Fanuc KAREL source: CE0115.KL

-- PROVISIONAL review KL for V770-1; original PC SHA256 38c2cadad195cee7491331c5a626b45bc0db98ebdebf5f674fdae5275aeffe66
-- Incomplete behavior may be omitted. Consult companion uncertainty JSON. Do not deploy.
PROGRAM CE0115
%NOLOCKGROUP
-- UNRESOLVED_LOCAL_POOL 6 cells at code offset 94; source declarations unknown
-- DIRECT_LOCAL_WORD_ACCESS alone does not prove INTEGER, REAL, or BOOLEAN
BEGIN
  -- UNRESOLVED_PC offsets 0-1; opcodes 7B
  -- UNRESOLVED_PC offsets 6-16; opcodes 2D,7F
  -- UNRESOLVED_PC offsets 21-26; opcodes 7F,7B
  -- UNRESOLVED_PC offsets 31-43; opcodes 2D,9D,52,7F
  -- UNRESOLVED_PC offsets 48-53; opcodes 7F,7B
  -- UNRESOLVED_PC offsets 58-74; opcodes 2D,2E,69,7F
  -- UNRESOLVED_PC offsets 79-99; opcodes 7F,2B,2C,7B
  -- UNRESOLVED_PC offsets 104-115; opcodes 2E,23
  -- UNRESOLVED_PC offsets 120-131; opcodes 2E,23
  -- UNRESOLVED_PC offsets 136-147; opcodes 2E,23
  -- UNRESOLVED_PC offsets 152-163; opcodes 2E,23
  -- UNRESOLVED_PC offsets 168-175; opcodes 9D,23
  -- UNRESOLVED_PC offsets 180-187; opcodes 9C,23
  -- UNRESOLVED_PC offsets 192-202; opcodes 3F,75
  -- UNRESOLVED_PC offsets 207-217; opcodes 3F,75
  -- UNRESOLVED_PC offsets 222-236; opcodes 2E,22,9D,33,35
  -- UNRESOLVED_PC offsets 241-259; opcodes 2E,22,2E,33,35
  -- UNRESOLVED_PC offsets 264-282; opcodes 73,73,88,79
  -- UNRESOLVED_PC offsets 287-301; opcodes 21,9D,52,23
  -- UNRESOLVED_PC offsets 306-311; opcodes 7A
  -- UNRESOLVED_PC offsets 316-334; opcodes 21,2E,52,23
  -- UNRESOLVED_PC offsets 344-348; opcodes 7F
  -- UNRESOLVED_PC offsets 353-357; opcodes 27,AA
  -- UNRESOLVED_PC offsets 362-366; opcodes 7F
END CE0115
